Omron CX-Programmer project НовыйПроект (CX-Programmer 9.61)

# PLC Svetofor: CP1L-E EM

## Global symbols (name address type ; comment)
T0000 BOOL  ; красный
T0001 BOOL  ; красный + желтый
T0002 BOOL  ; зеленый
T0003 BOOL  ; зеленый мигающий
T0004 BOOL  ; желтый
T0005 BOOL  ; желтый вкл
T0006 BOOL  ; желтый выкл
T0007 BOOL  ; зеленый вкл
T0008 BOOL  ; зеленый выкл
W5 CHANNEL  ; Время * 10
Visible W0.00 BOOL  ; Отображение времени
add W2 UINT  ; Время фазы
green 100.02 BOOL  ; зеленый
red 100.00 BOOL  ; красный
run 0.00 BOOL  ; работа
t_green H1 UINT  ; время зеленого 0,1с
t_red H0 UINT  ; время красного 0,1с
yellow 100.01 BOOL  ; желтый
Блок_5 Функциональный_блок_5

## Program НоваяЗадача1 (cyclic task 0)
Local symbols
E 0.00 BOOL
F 0.01 BOOL
G 0.02 BOOL
H 0.03 BOOL
Y1 100.04 BOOL
YO 100.05 BOOL
a D10 INT
b D11 INT
button 0.06 BOOL
button1 0.07 BOOL
button2 0.11 BOOL
c D12 INT
d D13 INT
run1 0.01 BOOL
run2 0.02 BOOL
run3 0.03 BOOL
start 0.10 BOOL
start2 0.11 BOOL
x D14 INT

### Section Сегмент1

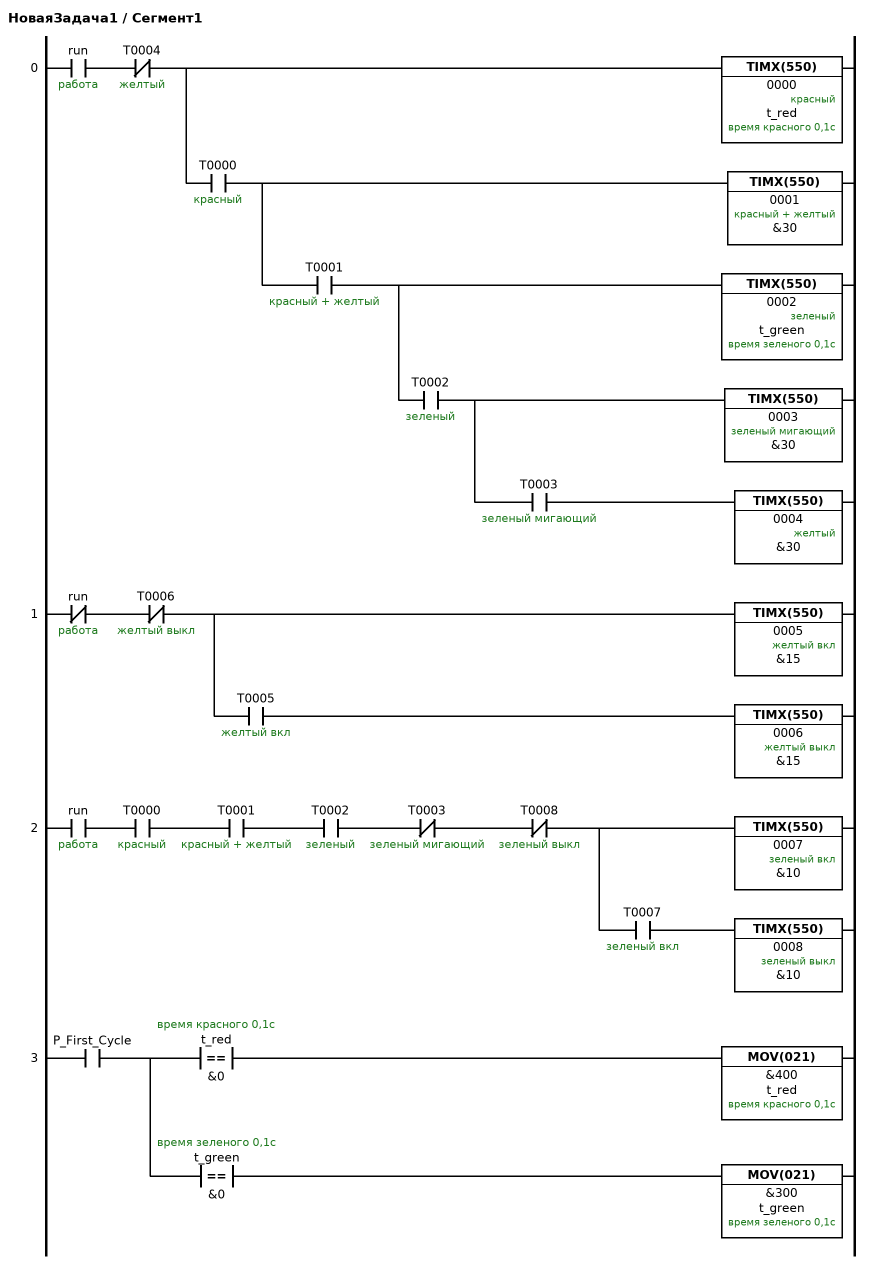
; rung 0
LD run  ; работа
ANDNOT T0004  ; желтый
TIMX(550) 0000 t_red  ; время красного 0,1с, красный
AND T0000  ; красный
TIMX(550) 0001 &30  ; красный + желтый
AND T0001  ; красный + желтый
TIMX(550) 0002 t_green  ; время зеленого 0,1с, зеленый
AND T0002  ; зеленый
TIMX(550) 0003 &30  ; зеленый мигающий
AND T0003  ; зеленый мигающий
TIMX(550) 0004 &30  ; желтый
; rung 1
LDNOT run  ; работа
ANDNOT T0006  ; желтый выкл
TIMX(550) 0005 &15  ; желтый вкл
AND T0005  ; желтый вкл
TIMX(550) 0006 &15  ; желтый выкл
; rung 2
LD run  ; работа
AND T0000  ; красный
AND T0001  ; красный + желтый
AND T0002  ; зеленый
ANDNOT T0003  ; зеленый мигающий
ANDNOT T0008  ; зеленый выкл
TIMX(550) 0007 &10  ; зеленый вкл
AND T0007  ; зеленый вкл
TIMX(550) 0008 &10  ; зеленый выкл
; rung 3
LD P_First_Cycle
OUT TR0
AND=(300) t_red &0  ; время красного 0,1с
MOV(021) &400 t_red  ; время красного 0,1с
LD TR0
AND=(300) t_green &0  ; время зеленого 0,1с
MOV(021) &300 t_green  ; время зеленого 0,1с

### Section Сегмент_2_0

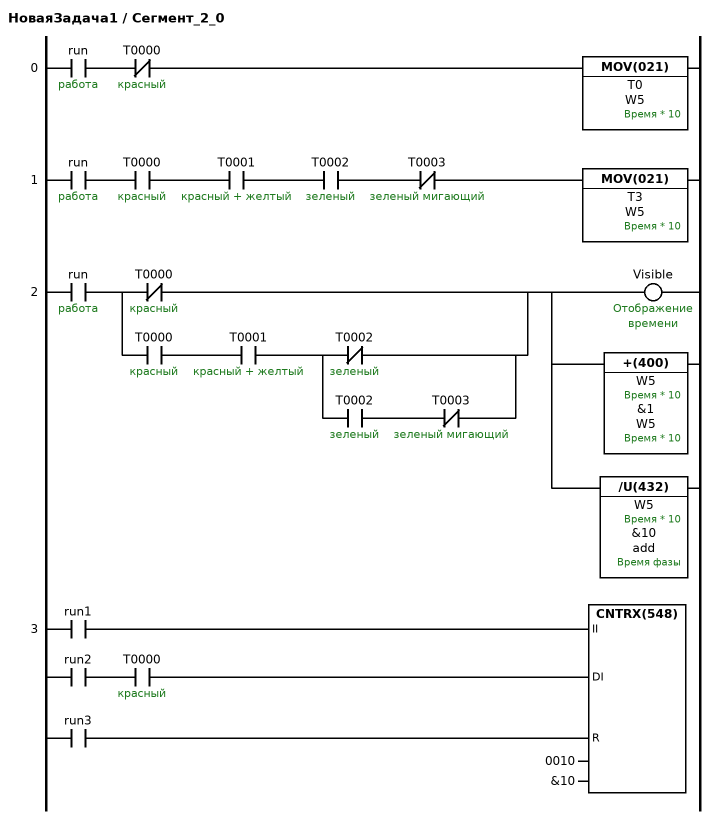
; rung 0
LD run  ; работа
ANDNOT T0000  ; красный
MOV(021) T0 W5  ; Время * 10
; rung 1
LD run  ; работа
AND T0000  ; красный
AND T0001  ; красный + желтый
AND T0002  ; зеленый
ANDNOT T0003  ; зеленый мигающий
MOV(021) T3 W5  ; Время * 10
; rung 2
LD run  ; работа
LDNOT T0000  ; красный
LD T0000  ; красный
AND T0001  ; красный + желтый
LDNOT T0002  ; зеленый
LD T0002  ; зеленый
ANDNOT T0003  ; зеленый мигающий
ORLD
ANDLD
ORLD
ANDLD
OUT Visible  ; Отображение времени
+(400) W5 &1 W5  ; Время * 10
/U(432) W5 &10 add  ; Время * 10, Время фазы
; rung 3
LD run1
LD run2
AND T0000  ; красный
LD run3
CNTRX(548) 0010 &10

### Section Сегмент3

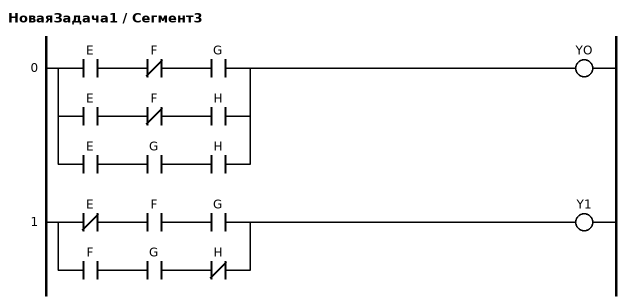
; rung 0
LD E
ANDNOT F
AND G
LD E
ANDNOT F
AND H
ORLD
LD E
AND G
AND H
ORLD
OUT YO
; rung 1
LDNOT E
AND F
AND G
LD F
AND G
ANDNOT H
ORLD
OUT Y1

### Section Сегмент_5

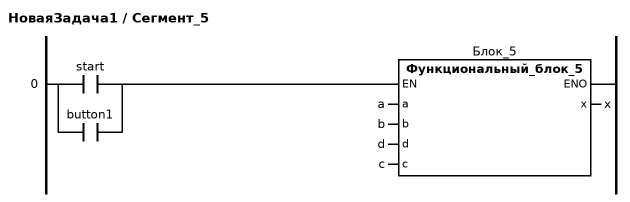
; rung 0
LD start
OR button1
CALL Блок_5 : Функциональный_блок_5 (a := a, b := b, d := d, c := c, x => x)

### Section Сегмент_51

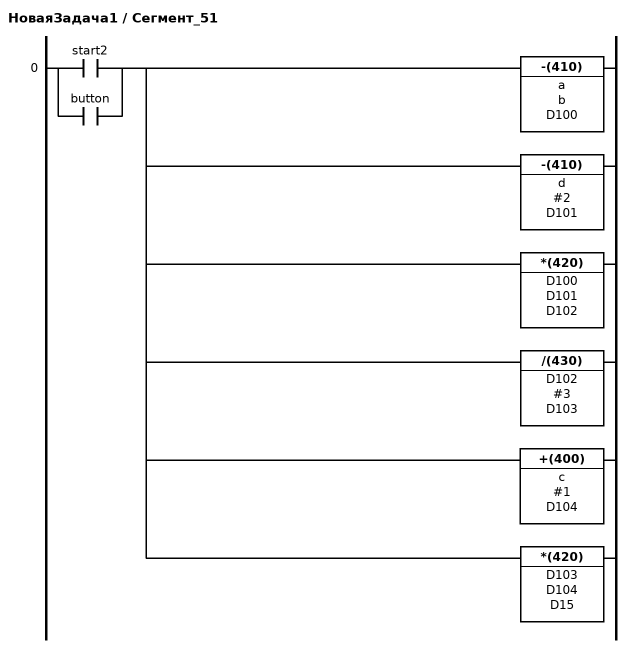
; rung 0
LD start2
OR button
-(410) a b D100
-(410) d #2 D101
*(420) D100 D101 D102
/(430) D102 #3 D103
+(400) c #1 D104
*(420) D103 D104 D15

### Section END
; rung 0
END(001)

## Function block Функциональный_блок_5
VAR_INPUT
  a : INT;
  b : INT;
  d : INT;
  c : INT;
END_VAR
VAR_OUTPUT
  x : INT;
END_VAR
x:=((a - b) * (d - 2)) / 3*(c + 1);

## Function block Функциональный_блок_51